FUNCTION F_UpdateEventTimestampWithSystemTime
VAR_INPUT
	stEvent : REFERENCE TO ST_Event;
END_VAR
VAR
	fbGETSYSTEMTIME : GETSYSTEMTIME;
	stFileTime : T_FILETIME;
END_VAR

fbGETSYSTEMTIME(timeLoDW => stFileTime.dwLowDateTime,
				timeHiDW => stFileTime.dwHighDateTime);

stEvent.dtTimestamp := FILETIME_TO_DT(fileTime := stFileTime);

END_FUNCTION

(* stored: Version 1.1.0.1, ProductVersion 3.1.4024.15
   POU F_UpdateEventTimestampWithSystemTime: Id {108e82b8-77b5-4d7c-9750-43190c973113}, SpecialFunc None *)
